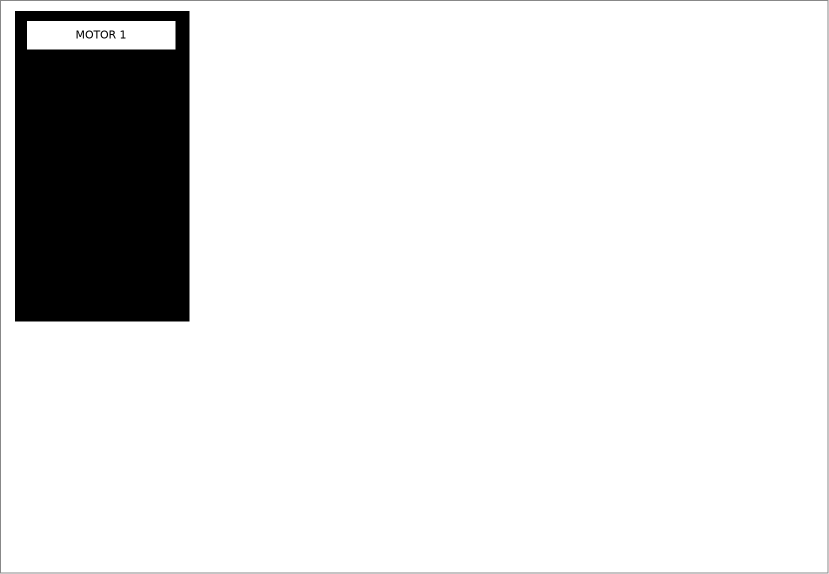
VISUALIZATION rotationControl  // 829x574
    Rectangle (15,11 174x310)
    Rectangle (26,20 150x30), "MOTOR 1"
END_VISUALIZATION

(* stored: Version 1.1.0.1, ProductVersion 3.1.4024.15
   Visu rotationControl: Id {5a72516b-b694-4179-bccd-2db7fa2d7720} *)
